INTERFACE ITF_TopElement1_HMI_Init EXTENDS ITF_BaseTopElement, ITF_TopElement1_HMI_Connector

END_INTERFACE

(* stored: Version 1.1.0.1
   Itf ITF_TopElement1_HMI_Init: Id {804f1863-12c9-0ab8-1a56-3b246519ba94} *)
